# B&R Automation Studio project TD52 (part 81)

#### rtwtypes.h
```c
/********************************************************************
 * COPYRIGHT -- B&R Industrial Automation GmbH
 ********************************************************************
 * Program: TrStRed
 * File: rtwtypes.h
 * Author: 105055527
 * Last modified by: maranen00
 * Created: Mon Sep 05 18:14:57 2016
 * Last modified: Mon Dec 06 12:59:10 2021
 * Model Version: 0.3.0
 * Description: Thermal reactor start time reduction function

   Outstandings:
   -------------
   - NA
 * modified Comment: V0.1.0 18.05.2021 Maran   TrStRed function first draft
   V0.1.1 27.05.2021 Maran   added limitation based on cyl. EG max temp. above setpoint
   V0.1.2 02.08.2021 Maran   added half load factor for function limit range
   V0.2.0 15.11.2021 Maran   added saturation limits to control error for the closed loop integrator (PERM parameters)
   V0.3.0 06.12.2021 Maran   removed unused logic in controller block; added filtered value of monitoring variables in debug interface
 ********************************************************************
 * Header for program TrStRed
 ********************************************************************
 * Generated with B&R Automation Studio Target for Simulink V6.3.1
 * (ERT based)
 ********************************************************************/

#ifndef RTWTYPES_H
#define RTWTYPES_H

/* Logical type definitions */
#if (!defined(__cplusplus))
#  ifndef false
#   define false                       (0U)
#  endif

#  ifndef true
#   define true                        (1U)
#  endif
#endif

/*=======================================================================*
 * Target hardware information
 *   Device type: Intel->x86/Pentium
 *   Number of bits:     char:   8    short:   16    long:  32
 *                       long:  32
 *                       native word size:  32
 *   Byte ordering: LittleEndian
 *   Signed integer division rounds to: Zero
 *   Shift right on a signed integer as arithmetic shift: on
 *=======================================================================*/

/*=======================================================================*
 * Fixed width word size data types:                                     *
 *   int8_T, int16_T, int32_T     - signed 8, 16, or 32 bit integers     *
 *   uint8_T, uint16_T, uint32_T  - unsigned 8, 16, or 32 bit integers   *
 *   real32_T, real64_T           - 32 and 64 bit floating point numbers *
 *=======================================================================*/
typedef signed char int8_T;
typedef unsigned char uint8_T;
typedef short int16_T;
typedef unsigned short uint16_T;
typedef long int32_T;
typedef unsigned long uint32_T;
typedef float real32_T;
typedef double real64_T;

/*===========================================================================*
 * Generic type definitions: boolean_T, char_T, byte_T, int_T, uint_T,       *
 *                           real_T, time_T, ulong_T.                        *
 *===========================================================================*/
typedef double real_T;
typedef double time_T;
typedef unsigned char boolean_T;
typedef long int_T;
typedef unsigned long uint_T;
typedef unsigned long ulong_T;
typedef char char_T;
typedef unsigned char uchar_T;
typedef char_T byte_T;

/*=======================================================================*
 * Min and Max:                                                          *
 *   int8_T, int16_T, int32_T     - signed 8, 16, or 32 bit integers     *
 *   uint8_T, uint16_T, uint32_T  - unsigned 8, 16, or 32 bit integers   *
 *=======================================================================*/
#define MAX_int8_T                     ((int8_T)(127))
#define MIN_int8_T                     ((int8_T)(-128))
#define MAX_uint8_T                    ((uint8_T)(255U))
#define MAX_int16_T                    ((int16_T)(32767))
#define MIN_int16_T                    ((int16_T)(-32768))
#define MAX_uint16_T                   ((uint16_T)(65535U))
#define MAX_int32_T                    ((int32_T)(2147483647))
#define MIN_int32_T                    ((int32_T)(-2147483647-1))
#define MAX_uint32_T                   ((uint32_T)(0xFFFFFFFFU))

/* Block D-Work pointer type */
typedef void * pointer_T;

#endif                                 /* RTWTYPES_H */

#ifndef MIN
#define MIN(a,b)                       ((a) < (b) ? (a) : (b))
#endif

#ifndef MAX
#define MAX(a,b)                       ((a) > (b) ? (a) : (b))
#endif

#ifndef AST_ROUND
#define AST_ROUND(x)                   ((x)>=0?(long long)((x)+0.5):(long long)((x)-0.5))
#endif
```

#### zero_crossing_types.h
```c
/********************************************************************
 * COPYRIGHT -- B&R Industrial Automation GmbH
 ********************************************************************
 * Program: TrStRed
 * File: zero_crossing_types.h
 * Author: 105055527
 * Last modified by: maranen00
 * Created: Mon Sep 05 18:14:57 2016
 * Last modified: Mon Dec 06 12:59:10 2021
 * Model Version: 0.3.0
 * Description: Thermal reactor start time reduction function

   Outstandings:
   -------------
   - NA
 * modified Comment: V0.1.0 18.05.2021 Maran   TrStRed function first draft
   V0.1.1 27.05.2021 Maran   added limitation based on cyl. EG max temp. above setpoint
   V0.1.2 02.08.2021 Maran   added half load factor for function limit range
   V0.2.0 15.11.2021 Maran   added saturation limits to control error for the closed loop integrator (PERM parameters)
   V0.3.0 06.12.2021 Maran   removed unused logic in controller block; added filtered value of monitoring variables in debug interface
 ********************************************************************
 * Header for program TrStRed
 ********************************************************************
 * Generated with B&R Automation Studio Target for Simulink V6.3.1
 * (ERT based)
 ********************************************************************/

#ifndef ZERO_CROSSING_TYPES_H
#define ZERO_CROSSING_TYPES_H
#include "rtwtypes.h"

/* Trigger directions: falling, either, and rising */
typedef enum {
  FALLING_ZERO_CROSSING = -1,
  ANY_ZERO_CROSSING = 0,
  RISING_ZERO_CROSSING = 1
} ZCDirection;

/* Previous state of a trigger signal */
typedef uint8_T ZCSigState;

/* Initial value of a trigger zero crossing signal */
#define UNINITIALIZED_ZCSIG            0x03U
#define NEG_ZCSIG                      0x02U
#define POS_ZCSIG                      0x01U
#define ZERO_ZCSIG                     0x00U

/* Current state of a trigger signal */
typedef enum {
  FALLING_ZCEVENT = -1,
  NO_ZCEVENT = 0,
  RISING_ZCEVENT = 1
} ZCEventType;

#endif                                 /* ZERO_CROSSING_TYPES_H */

#ifndef MIN
#define MIN(a,b)                       ((a) < (b) ? (a) : (b))
#endif

#ifndef MAX
#define MAX(a,b)                       ((a) > (b) ? (a) : (b))
#endif

#ifndef AST_ROUND
#define AST_ROUND(x)                   ((x)>=0?(long long)((x)+0.5):(long long)((x)-0.5))
#endif
```

### Library Logical/EngineController/Lib_EC/lSCRT_ss (ANSIC, version 1.00.0)

#### SCRT_ss.c
```c
/********************************************************************
 * COPYRIGHT -- B&R Industrial Automation GmbH
 ********************************************************************
 * Program: SCRT_ss
 * File: SCRT_ss.c
 * Author: 105055527
 * Last modified by: arnolge00
 * Created: Mon Sep 05 18:14:57 2016
 * Last modified: Fri Oct 01 08:40:23 2021
 * Model Version: 1.00
 * Description: Steady state detection for SCR inlet temperature controller vie ignition timing

   Outstandings:
   -------------
   - NA
 * modified Comment: V1.00  01.10.2021, Arnold, created
 ********************************************************************
 * Implementation of program SCRT_ss
 ********************************************************************
 * Generated with B&R Automation Studio Target for Simulink V6.3.0
 * (ERT based)
 ********************************************************************/

#include "SCRT_ss.h"
#include "SCRT_ss_private.h"

/*  Defines */

/*  Data Types */

/**************************** GLOBAL DATA *************************************/
/*  Definitions */

/*  Declarations  */

/***************************** FILE SCOPE DATA ********************************/

/*************************** FUNCTIONS ****************************************/

/* Model step function */
void SCRT_ss_step(RT_MODEL_SCRT_ss *const SCRT_ss_M, struct fSCRT_ss* inst)
{
  struct BlockIO_SCRT_ss *SCRT_ss_B = ((struct BlockIO_SCRT_ss *) SCRT_ss_M->blockIO);
  struct D_Work_SCRT_ss *SCRT_ss_DWork = ((struct D_Work_SCRT_ss *) SCRT_ss_M->dwork);
  ExternalOutputs_SCRT_ss *SCRT_ss_Y = (ExternalOutputs_SCRT_ss *)
    SCRT_ss_M->outputs;
  real32_T rtb_Switch_n;
  boolean_T rtb_LogicalOperator3;
  boolean_T rtb_LogicalOperator_f2;
  boolean_T rtb_LogicalOperator_m;
  boolean_T rtb_RelationalOperator;
  boolean_T rtb_LogicalOperator;
  boolean_T rtb_LogicalOperator2;
  real32_T tmp;

  /* S-Function (bur_bus_in): '<Root>/Bus Input2' */
  SCRT_ss_B->BusInput2 = inst->In;

  /* S-Function (bur_bus_in): '<Root>/Bus Input1' */
  SCRT_ss_B->BusInput1 = inst->Perm;

  /* Outputs for Atomic SubSystem: '<S4>/Filter' */
  /* RelationalOperator: '<S5>/Relational Operator' incorporates:
   *  Constant: '<S5>/Constant'
   *  Switch: '<S2>/Environment Switch'
   */
  rtb_LogicalOperator_f2 = (SCRT_ss_B->BusInput1.rTi_Filt_LXdev > 0.0F);

  /* End of Outputs for SubSystem: '<S4>/Filter' */

  /* Logic: '<S4>/NOT' incorporates:
   *  Logic: '<S4>/NOT1'
   *  Switch: '<S1>/Environment Switch'
   */
  rtb_LogicalOperator = !SCRT_ss_B->BusInput2.bEna;

  /* Outputs for Atomic SubSystem: '<S4>/Filter' */
  /* Logic: '<S5>/Logical Operator' incorporates:
   *  Logic: '<S4>/NOT'
   *  Logic: '<S5>/Logical Operator1'
   */
  rtb_LogicalOperator_m = (rtb_LogicalOperator || (!rtb_LogicalOperator_f2));

  /* DiscreteIntegrator: '<S5>/Discrete-Time Integrator' */
  if (rtb_LogicalOperator_m || (SCRT_ss_DWork->DiscreteTimeIntegrator_PrevRe_c
       != 0)) {
    SCRT_ss_DWork->DiscreteTimeIntegrator_DSTATE_f = 0.0F;
  }

  /* Switch: '<S5>/Switch' incorporates:
   *  DiscreteIntegrator: '<S5>/Discrete-Time Integrator'
   *  Switch: '<S1>/Environment Switch'
   */
  if (rtb_LogicalOperator_f2) {
    rtb_Switch_n = SCRT_ss_DWork->DiscreteTimeIntegrator_DSTATE_f;
  } else {
    rtb_Switch_n = SCRT_ss_B->BusInput2.rPr_Leanox_Dev;
  }

  /* End of Switch: '<S5>/Switch' */

  /* Switch: '<S8>/Switch' incorporates:
   *  Abs: '<S8>/Abs'
   *  RelationalOperator: '<S8>/Relational Operator'
   *  Switch: '<S2>/Environment Switch'
   */
  if (2.22044605E-16F >= (real32_T)fabs(SCRT_ss_B->BusInput1.rTi_Filt_LXdev)) {
    tmp = 2.22044605E-16F;
  } else {
    tmp = SCRT_ss_B->BusInput1.rTi_Filt_LXdev;
  }

  /* End of Switch: '<S8>/Switch' */

  /* Update for DiscreteIntegrator: '<S5>/Discrete-Time Integrator' incorporates:
   *  Product: '<S5>/Divide4'
   *  Sum: '<S5>/Sum4'
   *  Switch: '<S1>/Environment Switch'
   */
  SCRT_ss_DWork->DiscreteTimeIntegrator_DSTATE_f +=
    (SCRT_ss_B->BusInput2.rPr_Leanox_Dev -
     SCRT_ss_DWork->DiscreteTimeIntegrator_DSTATE_f) / tmp * 0.01F;
  SCRT_ss_DWork->DiscreteTimeIntegrator_PrevRe_c = (int8_T)rtb_LogicalOperator_m;

  /* End of Outputs for SubSystem: '<S4>/Filter' */

  /* RelationalOperator: '<S4>/Relational Operator' incorporates:
   *  Abs: '<S4>/Abs'
   *  Switch: '<S2>/Environment Switch'
   */
  rtb_LogicalOperator_m = ((real32_T)fabs(rtb_Switch_n) <=
    SCRT_ss_B->BusInput1.rThreshold_LXdev_ss);

  /* Outputs for Atomic SubSystem: '<S4>/Filter1' */
  /* RelationalOperator: '<S6>/Relational Operator' incorporates:
   *  Constant: '<S6>/Constant'
   *  Switch: '<S2>/Environment Switch'
   */
  rtb_LogicalOperator_f2 = (SCRT_ss_B->BusInput1.rTi_Filt_Pset > 0.0F);

  /* Logic: '<S6>/Logical Operator' incorporates:
   *  Logic: '<S6>/Logical Operator1'
   */
  rtb_LogicalOperator = (rtb_LogicalOperator || (!rtb_LogicalOperator_f2));

  /* DiscreteIntegrator: '<S6>/Discrete-Time Integrator' incorporates:
   *  Switch: '<S1>/Environment Switch'
   */
  if (SCRT_ss_DWork->DiscreteTimeIntegrator_IC_LOADI != 0) {
    SCRT_ss_DWork->DiscreteTimeIntegrator_DSTATE_e =
      SCRT_ss_B->BusInput2.rP_Set_Norm;
  }

  if (rtb_LogicalOperator || (SCRT_ss_DWork->DiscreteTimeIntegrator_PrevRe_g !=
       0)) {
    SCRT_ss_DWork->DiscreteTimeIntegrator_DSTATE_e =
      SCRT_ss_B->BusInput2.rP_Set_Norm;
  }

  /* Switch: '<S6>/Switch' incorporates:
   *  DiscreteIntegrator: '<S6>/Discrete-Time Integrator'
   *  Switch: '<S1>/Environment Switch'
   */
  if (rtb_LogicalOperator_f2) {
    rtb_Switch_n = SCRT_ss_DWork->DiscreteTimeIntegrator_DSTATE_e;
  } else {
    rtb_Switch_n = SCRT_ss_B->BusInput2.rP_Set_Norm;
  }

  /* End of Switch: '<S6>/Switch' */

  /* Update for DiscreteIntegrator: '<S6>/Discrete-Time Integrator' */
  SCRT_ss_DWork->DiscreteTimeIntegrator_IC_LOADI = 0U;

  /* Switch: '<S10>/Switch' incorporates:
   *  Abs: '<S10>/Abs'
   *  RelationalOperator: '<S10>/Relational Operator'
   *  Switch: '<S2>/Environment Switch'
   */
  if (2.22044605E-16F >= (real32_T)fabs(SCRT_ss_B->BusInput1.rTi_Filt_Pset)) {
    tmp = 2.22044605E-16F;
  } else {
    tmp = SCRT_ss_B->BusInput1.rTi_Filt_Pset;
  }

  /* End of Switch: '<S10>/Switch' */

  /* Update for DiscreteIntegrator: '<S6>/Discrete-Time Integrator' incorporates:
   *  Product: '<S6>/Divide4'
   *  Sum: '<S6>/Sum4'
   *  Switch: '<S1>/Environment Switch'
   */
  SCRT_ss_DWork->DiscreteTimeIntegrator_DSTATE_e +=
    (SCRT_ss_B->BusInput2.rP_Set_Norm -
     SCRT_ss_DWork->DiscreteTimeIntegrator_DSTATE_e) / tmp * 0.01F;
  SCRT_ss_DWork->DiscreteTimeIntegrator_PrevRe_g = (int8_T)rtb_LogicalOperator;

  /* End of Outputs for SubSystem: '<S4>/Filter1' */

  /* RelationalOperator: '<S4>/Relational Operator1' incorporates:
   *  Abs: '<S4>/Abs1'
   *  Sum: '<S4>/Sum'
   *  Switch: '<S1>/Environment Switch'
   *  Switch: '<S2>/Environment Switch'
   */
  rtb_LogicalOperator_f2 = ((real32_T)fabs(rtb_Switch_n -
    SCRT_ss_B->BusInput2.rP_Set_Norm) <= SCRT_ss_B->BusInput1.rThreshold_Pset_ss);

  /* Logic: '<S4>/AND' incorporates:
   *  Switch: '<S1>/Environment Switch'
   */
  rtb_LogicalOperator = (rtb_LogicalOperator_m && rtb_LogicalOperator_f2 &&
    SCRT_ss_B->BusInput2.bEna);

  /* Outputs for Atomic SubSystem: '<S4>/TON' */
  /* Logic: '<S7>/Logical Operator2' */
  rtb_LogicalOperator2 = !rtb_LogicalOperator;

  /* DiscreteIntegrator: '<S7>/Discrete-Time Integrator' */
  if (rtb_LogicalOperator2 || (SCRT_ss_DWork->DiscreteTimeIntegrator_PrevRese !=
       0)) {
    SCRT_ss_DWork->DiscreteTimeIntegrator_DSTATE = 0.0F;
  }

  /* RelationalOperator: '<S7>/Relational Operator' incorporates:
   *  DiscreteIntegrator: '<S7>/Discrete-Time Integrator'
   *  Switch: '<S2>/Environment Switch'
   */
  rtb_RelationalOperator = (SCRT_ss_DWork->DiscreteTimeIntegrator_DSTATE >=
    SCRT_ss_B->BusInput1.rTi_Delay_ss);

  /* Logic: '<S7>/Logical Operator3' */
  rtb_LogicalOperator3 = (rtb_RelationalOperator && rtb_LogicalOperator);

  /* Update for DiscreteIntegrator: '<S7>/Discrete-Time Integrator' incorporates:
   *  DataTypeConversion: '<S12>/Conversion'
   *  Logic: '<S7>/Logical Operator'
   *  Logic: '<S7>/Logical Operator1'
   */
  SCRT_ss_DWork->DiscreteTimeIntegrator_DSTATE += (real32_T)
    ((!rtb_RelationalOperator) && rtb_LogicalOperator) * 0.01F;
  SCRT_ss_DWork->DiscreteTimeIntegrator_PrevRese = (int8_T)rtb_LogicalOperator2;

  /* End of Outputs for SubSystem: '<S4>/TON' */

  /* Outport: '<Root>/Out' incorporates:
   *  BusCreator generated from: '<Root>/Out'
   */
  SCRT_ss_Y->Out.bSCRT_ss = rtb_LogicalOperator3;

  /* Outport: '<Root>/dbg' incorporates:
   *  BusCreator generated from: '<Root>/dbg'
   */
  SCRT_ss_Y->dbg.bss_LXdev = rtb_LogicalOperator_m;
  SCRT_ss_Y->dbg.bss_P = rtb_LogicalOperator_f2;
  SCRT_ss_Y->dbg.bss_noDelay = rtb_LogicalOperator;

  /* BusCreator generated from: '<Root>/Bus Output' */
  SCRT_ss_B->BusConversion_InsertedFor_BusOu.bSCRT_ss = rtb_LogicalOperator3;

  /* S-Function (bur_bus_out): '<Root>/Bus Output' */
  inst->Out = SCRT_ss_B->BusConversion_InsertedFor_BusOu;

  /* BusCreator generated from: '<Root>/Bus Output1' */
  SCRT_ss_B->BusConversion_InsertedFor_Bus_d.bss_LXdev = rtb_LogicalOperator_m;
  SCRT_ss_B->BusConversion_InsertedFor_Bus_d.bss_P = rtb_LogicalOperator_f2;
  SCRT_ss_B->BusConversion_InsertedFor_Bus_d.bss_noDelay = rtb_LogicalOperator;

  /* S-Function (bur_bus_out): '<Root>/Bus Output1' */
  inst->Dbg = SCRT_ss_B->BusConversion_InsertedFor_Bus_d;

  /* UnitDelay: '<S3>/Unit Delay' */
  SCRT_ss_B->UnitDelay = SCRT_ss_DWork->UnitDelay_DSTATE;

  /* S-Function (bur_out): '<Root>/Output1' */
  inst->Version = SCRT_ss_B->UnitDelay;

  /* Update for UnitDelay: '<S3>/Unit Delay' */
  SCRT_ss_DWork->UnitDelay_DSTATE = 100U;
}

/* Model initialize function */
void SCRT_ss_initialize(RT_MODEL_SCRT_ss *const SCRT_ss_M, struct fSCRT_ss* inst)
{
  struct D_Work_SCRT_ss *SCRT_ss_DWork = ((struct D_Work_SCRT_ss *) SCRT_ss_M->dwork);

  /* SystemInitialize for Atomic SubSystem: '<S4>/Filter1' */
  /* InitializeConditions for DiscreteIntegrator: '<S6>/Discrete-Time Integrator' */
  SCRT_ss_DWork->DiscreteTimeIntegrator_IC_LOADI = 1U;

  /* End of SystemInitialize for SubSystem: '<S4>/Filter1' */
}

/* Model terminate function */
void SCRT_ss_terminate(RT_MODEL_SCRT_ss *const SCRT_ss_M, struct fSCRT_ss* inst)
{
  /* (no terminate code required) */
  UNUSED_PARAMETER(SCRT_ss_M);
}

/*======================== TOOL VERSION INFORMATION ==========================*
 * MATLAB 9.8 (R2020a)18-Nov-2019                                             *
 * Simulink 10.1 (R2020a)18-Nov-2019                                          *
 * Simulink Coder 9.3 (R2020a)18-Nov-2019                                     *
 * Embedded Coder 7.4 (R2020a)18-Nov-2019                                     *
 * Stateflow 10.2 (R2020a)18-Nov-2019                                         *
 *============================================================================*/

/*======================= LICENSE IN USE INFORMATION =========================*
 * matlab                                                                     *
 * matlab_coder                                                               *
 * real-time_workshop                                                         *
 * rtw_embedded_coder                                                         *
 * simulink                                                                   *
 *============================================================================*/
```

#### SCRT_ss.h
```c
/********************************************************************
 * COPYRIGHT -- B&R Industrial Automation GmbH
 ********************************************************************
 * Program: SCRT_ss
 * File: SCRT_ss.h
 * Author: 105055527
 * Last modified by: arnolge00
 * Created: Mon Sep 05 18:14:57 2016
 * Last modified: Fri Oct 01 08:40:23 2021
 * Model Version: 1.00
 * Description: Steady state detection for SCR inlet temperature controller vie ignition timing

   Outstandings:
   -------------
   - NA
 * modified Comment: V1.00  01.10.2021, Arnold, created
 ********************************************************************
 * Header for program SCRT_ss
 ********************************************************************
 * Generated with B&R Automation Studio Target for Simulink V6.3.0
 * (ERT based)
 ********************************************************************/

#ifndef RTW_HEADER_SCRT_ss_h_
#define RTW_HEADER_SCRT_ss_h_
#include <math.h>
#ifndef SCRT_ss_COMMON_INCLUDES_
# define SCRT_ss_COMMON_INCLUDES_
#include "rtwtypes.h"
#endif                                 /* SCRT_ss_COMMON_INCLUDES_ */

#include "SCRT_ss_types.h"
#include "lSCRT_ss.h"
/* Beginning of Dynamic TypeDefs: */
/* End of Dynamic TypeDefs: */
#ifndef MIN
#define MIN(a,b)	((a) < (b) ? (a) : (b))
#endif

#ifndef MAX
#define MAX(a,b)	((a) > (b) ? (a) : (b))
#endif

#ifndef AST_ROUND
#define AST_ROUND(x) ((x)>=0?(long long)((x)+0.5):(long long)((x)-0.5))
#endif

#include "rt_defines.h"

/* Macros for accessing real-time model data structure */
#ifndef rtmGetBlockIO
# define rtmGetBlockIO(rtm)            ((rtm)->blockIO)
#endif

#ifndef rtmSetBlockIO
# define rtmSetBlockIO(rtm, val)       ((rtm)->blockIO = (val))
#endif

#ifndef rtmGetRootDWork
# define rtmGetRootDWork(rtm)          ((rtm)->dwork)
#endif

#ifndef rtmSetRootDWork
# define rtmSetRootDWork(rtm, val)     ((rtm)->dwork = (val))
#endif

#ifndef rtmGetU
# define rtmGetU(rtm)                  ((rtm)->inputs)
#endif

#ifndef rtmSetU
# define rtmSetU(rtm, val)             ((rtm)->inputs = (val))
#endif

#ifndef rtmGetY
# define rtmGetY(rtm)                  ((rtm)->outputs)
#endif

#ifndef rtmSetY
# define rtmSetY(rtm, val)             ((rtm)->outputs = (val))
#endif

#ifndef rtmGetErrorStatus
# define rtmGetErrorStatus(rtm)        ((rtm)->errorStatus)
#endif

#ifndef rtmSetErrorStatus
# define rtmSetErrorStatus(rtm, val)   ((rtm)->errorStatus = (val))
#endif

#ifndef MIN
#define MIN(a,b)                       ((a) < (b) ? (a) : (b))
#endif

#ifndef MAX
#define MAX(a,b)                       ((a) > (b) ? (a) : (b))
#endif

#ifndef AST_ROUND
#define AST_ROUND(x)                   ((x)>=0?(long long)((x)+0.5):(long long)((x)-0.5))
#endif

/* user code (top of header file) */
/***************************************************************************************************
 * COPYRIGHT -- INNIO Jenbacher GmbH & CO OG
 ****************************************************************************************************
 * Program:            Demo
 * Author:             arnolge00
 * Created:            03.04.2020 22:15
 ****************************************************************************************************
 * MODEL INFORMATION
 ****************************************************************************************************
 * Model Name:         C:\Users\arnolge00\Documents\MATLAB\Demo\Demo.slx
 * Model Version:      1.01
 * Simulink Version:   R2018b
 * B&R Target:         V6.1.0
 * Description:        Demo Version of two filters with additional signal quality check
 *
 *                     Outstandings:
 *                     -------------
 *                     - NA
 ****************************************************************************************************
 * HISTORY
 ****************************************************************************************************
 * Last Modified By:   arnolge00
 * Last Modified Date: Fri Apr 03 22:06:49 2020
 * Modified Comment:   V1.00  18.09.2018 Arnold   created for training
 *                     V1.01  19.09.2018 Arnold   test
 ****************************************************************************************************/

/* Block signals (default storage) */

/* Block states (default storage) for system '<Root>' */

/* External inputs (root inport signals with default storage) */

/* External outputs (root outports fed by signals with default storage) */

/* Real-time Model Data Structure */

/* Model entry point functions */
extern void SCRT_ss_initialize(RT_MODEL_SCRT_ss *const SCRT_ss_M, struct fSCRT_ss* inst);
extern void SCRT_ss_step(RT_MODEL_SCRT_ss *const SCRT_ss_M, struct fSCRT_ss* inst);
extern void SCRT_ss_terminate(RT_MODEL_SCRT_ss *const SCRT_ss_M, struct fSCRT_ss* inst);

/*-
 * The generated code includes comments that allow you to trace directly
 * back to the appropriate location in the model.  The basic format
 * is <system>/block_name, where system is the system number (uniquely
 * assigned by Simulink) and block_name is the name of the block.
 *
 * Use the MATLAB hilite_system command to trace the generated code back
 * to the model.  For example,
 *
 * hilite_system('<S3>')    - opens system 3
 * hilite_system('<S3>/Kp') - opens and selects block Kp which resides in S3
 *
 * Here is the system hierarchy for this model
 *
 * '<Root>' : 'SCRT_ss'
 * '<S1>'   : 'SCRT_ss/Environment Controller'
 * '<S2>'   : 'SCRT_ss/Environment Controller2'
 * '<S3>'   : 'SCRT_ss/Info'
 * '<S4>'   : 'SCRT_ss/SteadyState'
 * '<S5>'   : 'SCRT_ss/SteadyState/Filter'
 * '<S6>'   : 'SCRT_ss/SteadyState/Filter1'
 * '<S7>'   : 'SCRT_ss/SteadyState/TON'
 * '<S8>'   : 'SCRT_ss/SteadyState/Filter/Divisor'
 * '<S9>'   : 'SCRT_ss/SteadyState/Filter/Divisor/Data Type Conversion Inherited'
 * '<S10>'  : 'SCRT_ss/SteadyState/Filter1/Divisor'
 * '<S11>'  : 'SCRT_ss/SteadyState/Filter1/Divisor/Data Type Conversion Inherited'
 * '<S12>'  : 'SCRT_ss/SteadyState/TON/Data Type Conversion Inherited'
 */
#endif                                 /* RTW_HEADER_SCRT_ss_h_ */
```

#### SCRT_ss_private.h
```c
/********************************************************************
 * COPYRIGHT -- B&R Industrial Automation GmbH
 ********************************************************************
 * Program: SCRT_ss
 * File: SCRT_ss_private.h
 * Author: 105055527
 * Last modified by: arnolge00
 * Created: Mon Sep 05 18:14:57 2016
 * Last modified: Fri Oct 01 08:40:23 2021
 * Model Version: 1.00
 * Description: Steady state detection for SCR inlet temperature controller vie ignition timing

   Outstandings:
   -------------
   - NA
 * modified Comment: V1.00  01.10.2021, Arnold, created
 ********************************************************************
 * Header for program SCRT_ss
 ********************************************************************
 * Generated with B&R Automation Studio Target for Simulink V6.3.0
 * (ERT based)
 ********************************************************************/

#ifndef RTW_HEADER_SCRT_ss_private_h_
#define RTW_HEADER_SCRT_ss_private_h_
#include "rtwtypes.h"
#include <bur/plctypes.h>
#ifndef MIN
#define MIN(a,b)                       ((a) < (b) ? (a) : (b))
#endif

#ifndef MAX
#define MAX(a,b)                       ((a) > (b) ? (a) : (b))
#endif

#ifndef AST_ROUND
#define AST_ROUND(x)                   ((x)>=0?(long long)((x)+0.5):(long long)((x)-0.5))
#endif
#endif                                 /* RTW_HEADER_SCRT_ss_private_h_ */
```

#### SCRT_ss_types.h
```c
/********************************************************************
 * COPYRIGHT -- B&R Industrial Automation GmbH
 ********************************************************************
 * Program: SCRT_ss
 * File: SCRT_ss_types.h
 * Author: 105055527
 * Last modified by: arnolge00
 * Created: Mon Sep 05 18:14:57 2016
 * Last modified: Fri Oct 01 08:40:23 2021
 * Model Version: 1.00
 * Description: Steady state detection for SCR inlet temperature controller vie ignition timing

   Outstandings:
   -------------
   - NA
 * modified Comment: V1.00  01.10.2021, Arnold, created
 ********************************************************************
 * Header for program SCRT_ss
 ********************************************************************
 * Generated with B&R Automation Studio Target for Simulink V6.3.0
 * (ERT based)
 ********************************************************************/

#ifndef RTW_HEADER_SCRT_ss_types_h_
#define RTW_HEADER_SCRT_ss_types_h_
#include "rtwtypes.h"

/* Model Code Variants */
#ifndef MIN
#define MIN(a,b)                       ((a) < (b) ? (a) : (b))
#endif

#ifndef MAX
#define MAX(a,b)                       ((a) > (b) ? (a) : (b))
#endif

#ifndef AST_ROUND
#define AST_ROUND(x)                   ((x)>=0?(long long)((x)+0.5):(long long)((x)-0.5))
#endif

/* Forward declaration for rtModel */

#endif                                 /* RTW_HEADER_SCRT_ss_types_h_ */
```

#### fSCRT_ss.c
```c
/********************************************************************
 * COPYRIGHT -- B&R Industrial Automation GmbH
 ********************************************************************
 * Program: SCRT_ss
 * File: fSCRT_ss.c
 * Author: 105055527
 * Last modified by: arnolge00
 * Created: Mon Sep 05 18:14:57 2016
 * Last modified: Fri Oct 01 08:40:23 2021
 * Model Version: 1.00
 * Description: Steady state detection for SCR inlet temperature controller vie ignition timing

   Outstandings:
   -------------
   - NA
 * modified Comment: V1.00  01.10.2021, Arnold, created
 ********************************************************************
 * Implementation of program SCRT_ss
 ********************************************************************
 * Generated with B&R Automation Studio Target for Simulink V6.3.0
 * (ERT based)
 ********************************************************************/

#include <bur/plctypes.h>
#include "SCRT_ss.h"
#include "rtwtypes.h"

/* Defines */
#define SS_TERMINATE 4
#define SS_OUTPUT 3
#define SS_INITIALIZE 2

/*  Data Types */

/**************************** GLOBAL DATA *************************************/
/*  Definitions */

/*  Declarations  */

/***************************** FILE SCOPE DATA ********************************/

/*************************** FUNCTIONS ****************************************/
#ifdef __cplusplus

unsigned long bur_heap_size = 6553500;

#endif

/*LEGACYMODE_VARIABLES*/
void fSCRT_ss(struct fSCRT_ss* inst)
{
  tag_RTM_SCRT_ss* const SCRT_ss_M = &(inst)->bur_SCRT_ss;
	inst->bur_SCRT_ss.blockIO = &(inst)->bur_BlockIO_SCRT_ss;
	inst->bur_SCRT_ss.inputs = &(inst)->bur_ExternalInputs_SCRT_ss;
	inst->bur_SCRT_ss.outputs = &(inst)->bur_ExternalOutputs_SCRT_ss;
	inst->bur_SCRT_ss.dwork = &(inst)->bur_D_Work_SCRT_ss;

  switch (inst->ssMethodType)
  {
   case SS_INITIALIZE:
    /* call model initialize function */
    SCRT_ss_initialize(SCRT_ss_M, inst);
    break;

   case SS_OUTPUT:
    /* call model step function */
    SCRT_ss_step(SCRT_ss_M, inst);

    break;

   case SS_TERMINATE:
    /* call model terminate function */
    SCRT_ss_terminate(SCRT_ss_M, inst);
    break;
  }
}

/*****************************************************************************
   Function block sample time: 0.01s
 *****************************************************************************/

/*****************************************************************************
   B&R Automation Studio Target for Simulink Version: A6.3.0 (23-Oct-2020)
 *****************************************************************************/

/*======================== TOOL VERSION INFORMATION ==========================*
 * MATLAB 9.8 (R2020a)18-Nov-2019                                             *
 * Simulink 10.1 (R2020a)18-Nov-2019                                          *
 * Simulink Coder 9.3 (R2020a)18-Nov-2019                                     *
 * Embedded Coder 7.4 (R2020a)18-Nov-2019                                     *
 * Stateflow 10.2 (R2020a)18-Nov-2019                                         *
 *============================================================================*/

/*======================= LICENSE IN USE INFORMATION =========================*
 * matlab                                                                     *
 * matlab_coder                                                               *
 * real-time_workshop                                                         *
 * rtw_embedded_coder                                                         *
 * simulink                                                                   *
 *============================================================================*/
```

#### lSCRT_ss.fun
```iecst
FUNCTION_BLOCK fSCRT_ss
  VAR_INPUT
    ssMethodType: SINT;
  END_VAR
  VAR_INPUT
        In : SCRT_ss_IN_Bus; (**)
  END_VAR
  VAR_INPUT
        Perm : SCRT_ss_PERM_Bus; (**)
  END_VAR
  VAR_OUTPUT
        Out : SCRT_ss_OUT_Bus; (**)
  END_VAR
  VAR_OUTPUT
        Dbg : SCRT_ss_DBG_Bus; (**)
  END_VAR
  VAR_OUTPUT
        Version : UDINT; (**)
  END_VAR
	VAR
		bur_BlockIO_SCRT_ss : BlockIO_SCRT_ss;
	END_VAR
	VAR
		bur_ExternalInputs_SCRT_ss : ExternalInputs_SCRT_ss;
	END_VAR
	VAR
		bur_ExternalOutputs_SCRT_ss : ExternalOutputs_SCRT_ss;
	END_VAR
	VAR
		bur_D_Work_SCRT_ss : D_Work_SCRT_ss;
	END_VAR
	VAR
		bur_SCRT_ss : tag_RTM_SCRT_ss;
	END_VAR
END_FUNCTION_BLOCK
```

#### lSCRT_ss.typ
```iecst
TYPE
	SCRT_ss_DBG_Bus : 	STRUCT
		bss_LXdev : BOOL; (* ()*)
		bss_P : BOOL; (* ()*)
		bss_noDelay : BOOL; (* ()*)
	END_STRUCT;
	SCRT_ss_IN_Bus : 	STRUCT
		rP_Set_Norm : REAL; (*Reset filter (p.u.)*)
		rPr_Leanox_Dev : REAL; (*Leanox controller deviaition (bar)*)
		bEna : BOOL; (*Enable Feature ()*)
	END_STRUCT;
	SCRT_ss_OUT_Bus : 	STRUCT
		bSCRT_ss : BOOL; (*steady state ()*)
	END_STRUCT;
	SCRT_ss_PERM_Bus : 	STRUCT
		rTi_Filt_Pset : REAL; (*Filter time constant for power setpoint (sec)*)
		rTi_Filt_LXdev : REAL; (*Filter teime constatn for leanox deviation (sec)*)
		rThreshold_Pset_ss : REAL; (*steady state threshold Pset (p.u.)*)
		rThreshold_LXdev_ss : REAL; (*steady state threshold leanox deviation (bar)*)
		rTi_Delay_ss : REAL; (*steady state threshold leanox deviation (sec)*)
	END_STRUCT;
	BlockIO_SCRT_ss : 	STRUCT
		BusInput1 : SCRT_ss_PERM_Bus;
		BusInput2 : SCRT_ss_IN_Bus;
		BusConversion_InsertedFor_BusOu : SCRT_ss_OUT_Bus;
		BusConversion_InsertedFor_Bus_d : SCRT_ss_DBG_Bus;
		UnitDelay : UDINT;
	END_STRUCT;
	D_Work_SCRT_ss : 	STRUCT
		DiscreteTimeIntegrator_DSTATE : REAL;
		DiscreteTimeIntegrator_DSTATE_e : REAL;
		DiscreteTimeIntegrator_DSTATE_f : REAL;
		UnitDelay_DSTATE : UDINT;
		DiscreteTimeIntegrator_PrevRese : SINT;
		DiscreteTimeIntegrator_PrevRe_g : SINT;
		DiscreteTimeIntegrator_PrevRe_c : SINT;
		DiscreteTimeIntegrator_IC_LOADI : USINT;
	END_STRUCT;
	ExternalInputs_SCRT_ss : 	STRUCT
		In : SCRT_ss_IN_Bus;
		Perm : SCRT_ss_PERM_Bus;
	END_STRUCT;
	ExternalOutputs_SCRT_ss : 	STRUCT
		Out : SCRT_ss_OUT_Bus;
		dbg : SCRT_ss_DBG_Bus;
	END_STRUCT;
	tag_RTM_SCRT_ss : 	STRUCT
		errorStatus : REFERENCE TO USINT;
		blockIO : REFERENCE TO BlockIO_SCRT_ss;
		inputs : REFERENCE TO ExternalInputs_SCRT_ss;
		outputs : REFERENCE TO ExternalOutputs_SCRT_ss;
		dwork : REFERENCE TO D_Work_SCRT_ss;
	END_STRUCT;
	RT_MODEL_SCRT_ss :tag_RTM_SCRT_ss;
END_TYPE
```

#### lib_properties.txt
```
For manual assignment to hardware configuration please
add the following additional include directories:

\Logical\MATLAB_includes\R2020a\

And the following additional build options:

-lm -D MODEL=SCRT_ss -D NUMST=1 -D NCSTATES=0 -D HAVESTDIO -D MODEL_HAS_DYNAMICALLY_LOADED_SFCNS=0 -D CLASSIC_INTERFACE=0 -D ALLOCATIONFCN=0 -D TID01EQ=0 -D TERMFCN=1 -D ONESTEPFCN=1 -D MAT_FILE=0 -D MULTI_INSTANCE_CODE=1 -D INTEGER_CODE=0 -D MT=0
```

#### rt_defines.h
```c
/********************************************************************
 * COPYRIGHT -- B&R Industrial Automation GmbH
 ********************************************************************
 * Program: SCRT_ss
 * File: rt_defines.h
 * Author: 105055527
 * Last modified by: arnolge00
 * Created: Mon Sep 05 18:14:57 2016
 * Last modified: Fri Oct 01 08:40:23 2021
 * Model Version: 1.00
 * Description: Steady state detection for SCR inlet temperature controller vie ignition timing

   Outstandings:
   -------------
   - NA
 * modified Comment: V1.00  01.10.2021, Arnold, created
 ********************************************************************
 * Header for program SCRT_ss
 ********************************************************************
 * Generated with B&R Automation Studio Target for Simulink V6.3.0
 * (ERT based)
 ********************************************************************/

#ifndef RTW_HEADER_rt_defines_h_
#define RTW_HEADER_rt_defines_h_
#ifndef MIN
#define MIN(a,b)                       ((a) < (b) ? (a) : (b))
#endif

#ifndef MAX
#define MAX(a,b)                       ((a) > (b) ? (a) : (b))
#endif

#ifndef AST_ROUND
#define AST_ROUND(x)                   ((x)>=0?(long long)((x)+0.5):(long long)((x)-0.5))
#endif

/*===========*
 * Constants *
 *===========*/
#define RT_PI                          3.14159265358979323846
#define RT_PIF                         3.1415927F
#define RT_LN_10                       2.30258509299404568402
#define RT_LN_10F                      2.3025851F
#define RT_LOG10E                      0.43429448190325182765
#define RT_LOG10EF                     0.43429449F
#define RT_E                           2.7182818284590452354
#define RT_EF                          2.7182817F

/*
 * UNUSED_PARAMETER(x)
 *   Used to specify that a function parameter (argument) is required but not
 *   accessed by the function body.
 */
#ifndef UNUSED_PARAMETER
# if defined(__LCC__)
#   define UNUSED_PARAMETER(x)                                   /* do nothing */
# else

/*
 * This is the semi-ANSI standard way of indicating that an
 * unused function parameter is required.
 */
#   define UNUSED_PARAMETER(x)         (void) (x)
# endif
#endif
#endif                                 /* RTW_HEADER_rt_defines_h_ */
```

#### rtwtypes.h
```c
/********************************************************************
 * COPYRIGHT -- B&R Industrial Automation GmbH
 ********************************************************************
 * Program: SCRT_ss
 * File: rtwtypes.h
 * Author: 105055527
 * Last modified by: arnolge00
 * Created: Mon Sep 05 18:14:57 2016
 * Last modified: Fri Oct 01 08:40:23 2021
 * Model Version: 1.00
 * Description: Steady state detection for SCR inlet temperature controller vie ignition timing

   Outstandings:
   -------------
   - NA
 * modified Comment: V1.00  01.10.2021, Arnold, created
 ********************************************************************
 * Header for program SCRT_ss
 ********************************************************************
 * Generated with B&R Automation Studio Target for Simulink V6.3.0
 * (ERT based)
 ********************************************************************/

#ifndef RTWTYPES_H
#define RTWTYPES_H

/* Logical type definitions */
#if (!defined(__cplusplus))
#  ifndef false
#   define false                       (0U)
#  endif

#  ifndef true
#   define true                        (1U)
#  endif
#endif

/*=======================================================================*
 * Target hardware information
 *   Device type: Intel->x86/Pentium
 *   Number of bits:     char:   8    short:   16    long:  32
 *                       long:  32
 *                       native word size:  32
 *   Byte ordering: LittleEndian
 *   Signed integer division rounds to: Zero
 *   Shift right on a signed integer as arithmetic shift: on
 *=======================================================================*/

/*=======================================================================*
 * Fixed width word size data types:                                     *
 *   int8_T, int16_T, int32_T     - signed 8, 16, or 32 bit integers     *
 *   uint8_T, uint16_T, uint32_T  - unsigned 8, 16, or 32 bit integers   *
 *   real32_T, real64_T           - 32 and 64 bit floating point numbers *
 *=======================================================================*/
typedef signed char int8_T;
typedef unsigned char uint8_T;
typedef short int16_T;
typedef unsigned short uint16_T;
typedef long int32_T;
typedef unsigned long uint32_T;
typedef float real32_T;
typedef double real64_T;

/*===========================================================================*
 * Generic type definitions: boolean_T, char_T, byte_T, int_T, uint_T,       *
 *                           real_T, time_T, ulong_T.                        *
 *===========================================================================*/
typedef double real_T;
typedef double time_T;
typedef unsigned char boolean_T;
typedef long int_T;
typedef unsigned long uint_T;
typedef unsigned long ulong_T;
typedef char char_T;
typedef unsigned char uchar_T;
typedef char_T byte_T;

/*=======================================================================*
 * Min and Max:                                                          *
 *   int8_T, int16_T, int32_T     - signed 8, 16, or 32 bit integers     *
 *   uint8_T, uint16_T, uint32_T  - unsigned 8, 16, or 32 bit integers   *
 *=======================================================================*/
#define MAX_int8_T                     ((int8_T)(127))
#define MIN_int8_T                     ((int8_T)(-128))
#define MAX_uint8_T                    ((uint8_T)(255U))
#define MAX_int16_T                    ((int16_T)(32767))
#define MIN_int16_T                    ((int16_T)(-32768))
#define MAX_uint16_T                   ((uint16_T)(65535U))
#define MAX_int32_T                    ((int32_T)(2147483647))
#define MIN_int32_T                    ((int32_T)(-2147483647-1))
#define MAX_uint32_T                   ((uint32_T)(0xFFFFFFFFU))

/* Block D-Work pointer type */
typedef void * pointer_T;

#endif                                 /* RTWTYPES_H */

#ifndef MIN
#define MIN(a,b)                       ((a) < (b) ? (a) : (b))
#endif

#ifndef MAX
#define MAX(a,b)                       ((a) > (b) ? (a) : (b))
#endif

#ifndef AST_ROUND
#define AST_ROUND(x)                   ((x)>=0?(long long)((x)+0.5):(long long)((x)-0.5))
#endif
```

### Library Logical/EngineController/Lib_EC/lGridStat (ANSIC, version 1.00.0)
